(* Logix 5000 project; controller cal1615 1756-L62 rev 20.19; software revision 20.05; part 81 of 81 *)
(* tags used below, declared in another part *)
   A00 : ALIAS FOR hmi_dint[0].0;
   A12 : ALIAS FOR hmi_dint[0].12;
   A30 : ALIAS FOR hmi_dint[0].30;
   accum_filling_on : ALIAS FOR hmi_dint[9].12;
   accum_holding_pressure_on : BOOL;   // Accumulator Holding Pressure Active
   add_sys_ramp : sys_Ramp;   // Addon Ramp
   ai_lpt01_pct : REAL;   // AI: Linear Position Transducer [%]
   ao_prs01 : REAL;   // AO: Pressure 1
   ao_prs02 : REAL;   // AO: Pressure 2
   control_to_empty : ALIAS FOR hmi_dint[9].13;
   di_ss_close_nip : ALIAS FOR p00_io_winder:5:I.14;
   di_ss_nip_auto : ALIAS FOR p00_io_winder:5:I.13;
   do_carriage_lift_sol : ALIAS FOR p00_io_winder:4:O.7;
   do_close_nip_sol : ALIAS FOR p00_io_winder:4:O.8;
   do_nip_illuminated_ss : ALIAS FOR p00_io_winder:4:O.6;
   enable_control : BOOL;   // Accumulator - Enable Control
   filling_pressure : REAL;   // Accumulator Fill Pressure Tare + Tension + Fill PID Offset
   Me : ALIAS FOR p00_wac;
   nip_auto_open_request : BOOL;   // Nip Auto Open Request
   nip_close_request : ALIAS FOR hmi_dint[9].7;
   nip_mode_auto : BOOL;   // Nip Mode Auto
   nip_open_dwell : TIMER;   // Nip Roll Open Dwell Payout must be established before the nip lets go
   nip_open_request : BOOL;   // Nip Open Request
   nip_open_selected : BOOL;   // Nip Selector in OPEN Neither Auto nor Close
   oneshot : DINT;
   param_acc_empty_hyst : REAL;   // Parameter Accumulator Empty Hysteresis Re-engages this far above param_acc_empty_pct so the handover cannot chatter [% o
   param_acc_empty_pct : REAL;   // Parameter Accumulator Empty Pressure bleeds to param_prs_empty and the winder hands back to load cell tension control at
   param_acc_min_limit : REAL;   // Parameter Accumulator Low Min Limimt
   param_accel_rate : REAL;   // Parameter Acceleration Rate
   param_counter_prs : REAL;   // Parameter Counter Pressure
   param_decel_rate : REAL;   // Parameter Decleration Rate
   param_press_slope_empty : REAL;   // Parameter Pressure Curve Slope - BOTH DIRECTIONS Measured on the machine: 62.9 psi gave 30 lbf, 68.0 psi gave 46 lbf (46
   param_prs_empty : REAL;   // Parameter Accumulator Pressure - EMPTY Bled out, carriage on the bottom stop, adds no tension [psi]
   param_prs_fill : REAL;   // Parameter RETIRED - fill pressure is calculated now See filling_pressure [psi]
   param_prs_payout : REAL;   // Parameter RETIRED - payout pressure is calculated now See wac_tension_pressure [psi]
   param_tare_pressure : REAL;   // Parameter Zero-Tension Pressure - PAYING OUT 62.9 - 30/3.14 = 53.4 [psi]
   param_tare_pressure_fill : REAL;   // Parameter Zero-Tension Pressure - FILLING Higher than paying out because friction reverses sign 83 psi held 70 lbf while
   pb_acc_on : ALIAS FOR hmi_dint[9].2;
   request_fill : ALIAS FOR hmi_dint[9].1;
   selected_pressure : REAL;   // Accumulator Selected Tension Pressure
   task_scan_time : REAL;   // Task Scan Time
   task_scan_time_dint : DINT;   // Task Scan
   timer_nip_open_delay : TIMER;   // Nip Open Dwell Timer
   W00 : ALIAS FOR hmi_dint[2].0;
   wac_tension_pressure : REAL;   // Winder Accumulator Tare + Web Tension Pressure Carriage Holds Position at Commanded Tension
   FAULT : BOOL;   // Fault AFI
   HMI : BOOL;   // AFI HMI
   nip_mode_close : BOOL;   // Nip Mode Close
   p00_FlashBit_1Sec : BOOL;   // System Flash Bit 1 Second
   p00_pb_lamp_test : BOOL;
   p00_wac : Accumulator;   // Winder Accumulator
   p00_wac_enabled : BOOL;   // Winder Accumulator Enabled Carriage lift on and pressure commanded Controls which loop holds web tension
   p00_wac_position_pct : REAL;   // Winder Accumulator Carriage Position Filtered [% of Stroke]
   p01_recipe_active : recipe;   // Active Recipe
   p01r09 : routine;   // System Modes
   p01r12_zero_line_speed : BOOL;   // System Line Accel Decel Control Line Speed at Zero
   p29_param_wind_out_stop_pct : REAL;   // Winder Wind Out Stop When the Accumulator Reaches This Position [% of Stroke]
   p29r15_request_run : BOOL;   // Winder Winder A VFD Request Run
   p29r16_request_run : BOOL;   // Winder Winder B VFD Request Run
(* P31_WAC, continued *)

ROUTINE R11_Modes   (* ladder *)
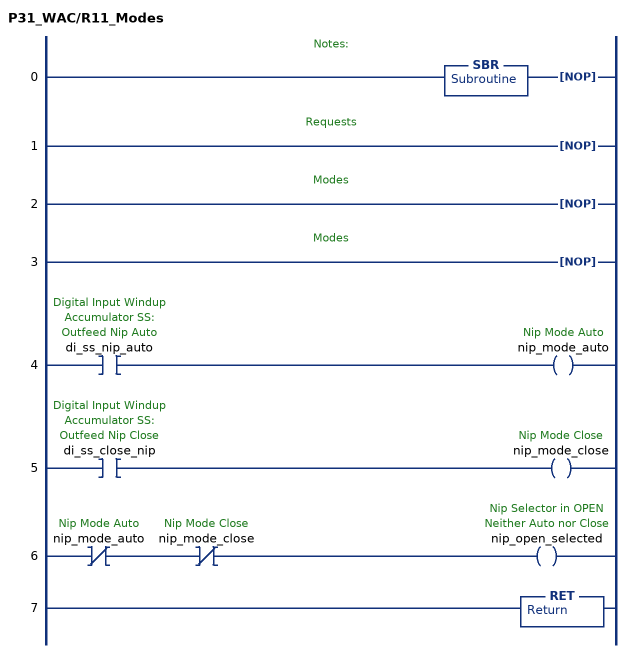
   // Notes:
   0: SBR()NOP();
   // Requests
   1: NOP();
   // Modes
   2: NOP();
   // Modes
   3: NOP();
   4: XIC(di_ss_nip_auto)OTE(nip_mode_auto);
   5: XIC(di_ss_close_nip)OTE(nip_mode_close);
   6: XIO(nip_mode_auto)XIO(nip_mode_close)OTE(nip_open_selected);
   7: RET();
END_ROUTINE

ROUTINE R21_Fill_Request   (* ladder *)
// WAC
// Fill Request and Tension Enable
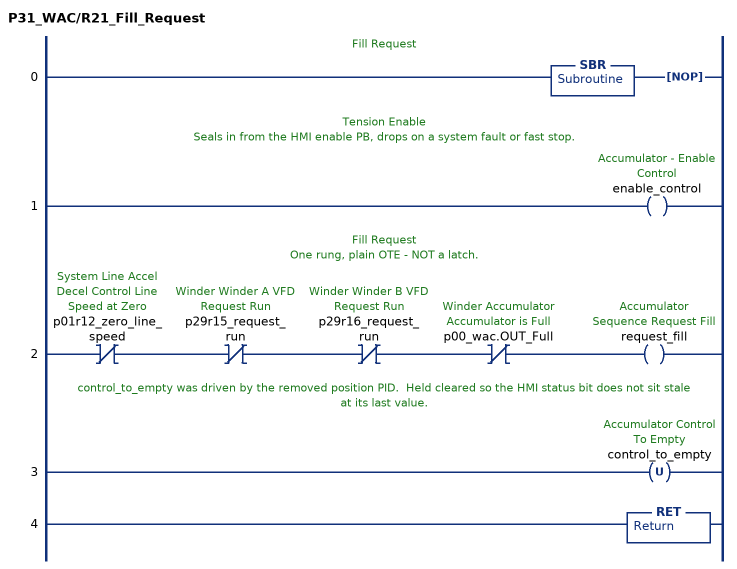
   // Fill Request
   0: SBR()NOP();
   // Tension Enable
   // Seals in from the HMI enable PB, drops on a system fault or fast stop.
   1: OTE(enable_control);
   // Fill Request
   // One rung, plain OTE - NOT a latch.
   2: XIO(p01r12_zero_line_speed)XIO(p29r15_request_run)XIO(p29r16_request_run)XIO(p00_wac.OUT_Full)OTE(request_fill);
   // control_to_empty was driven by the removed position PID.  Held cleared so the HMI status bit does not sit stale at its last value.
   3: OTU(control_to_empty);
   4: RET();
END_ROUTINE

ROUTINE R22_Fill_Pressure   (* ladder *)
// Windup Accumulator
// Fill Pressure
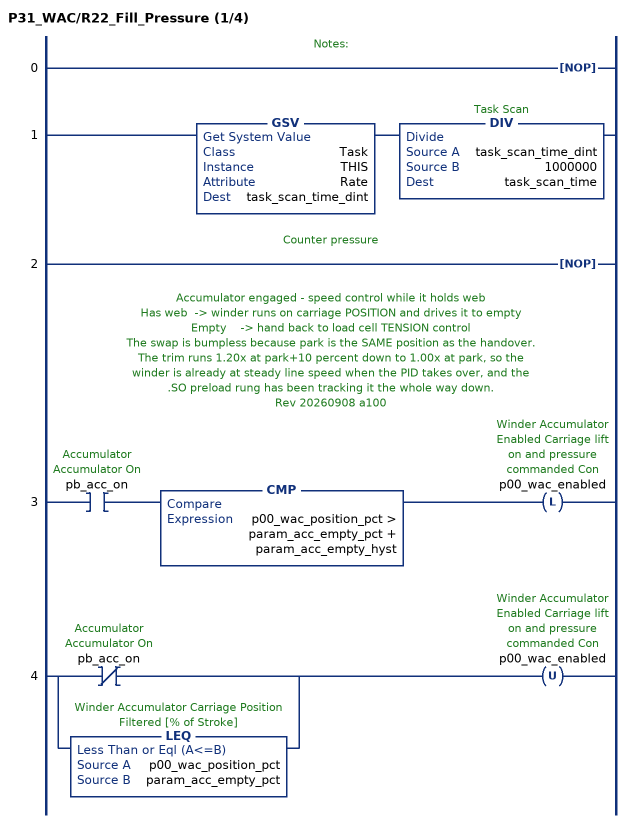
   // Notes:
   0: NOP();
   1: GSV(Task,THIS,Rate,task_scan_time_dint)DIV(task_scan_time_dint,1000000,task_scan_time);
   // Counter pressure
   2: NOP();
   // Accumulator engaged - speed control while it holds web
   // Has web  -> winder runs on carriage POSITION and drives it to empty
   // Empty    -> hand back to load cell TENSION control
   // The swap is bumpless because park is the SAME position as the handover.
   // The trim runs 1.20x at park+10 percent down to 1.00x at park, so the
   // winder is already at steady line speed when the PID takes over, and the
   // .SO preload rung has been tracking it the whole way down.
   // Rev 20260908 a100
   3: XIC(pb_acc_on)CMP(p00_wac_position_pct > param_acc_empty_pct + param_acc_empty_hyst)OTL(p00_wac_enabled);
   4: [XIO(pb_acc_on) ,LEQ(p00_wac_position_pct,param_acc_empty_pct) ]OTU(p00_wac_enabled);
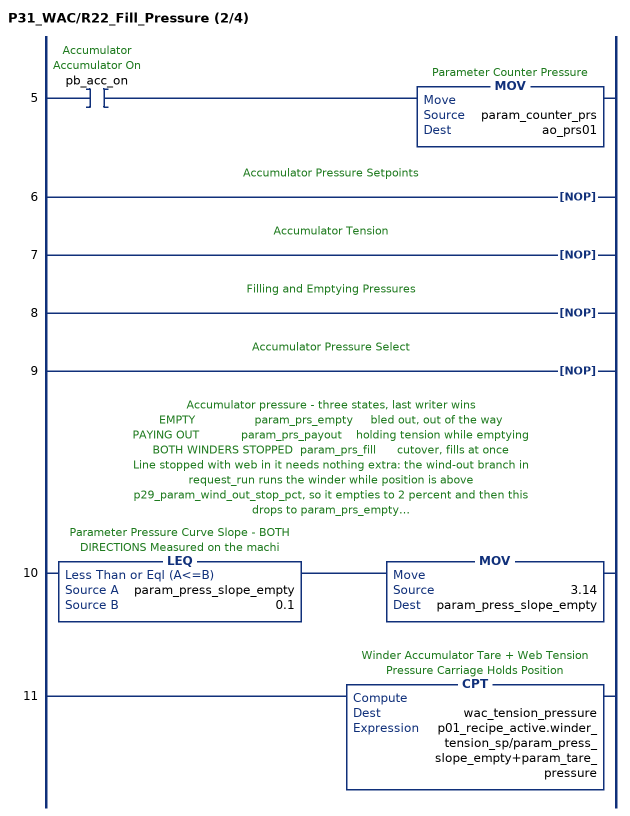
   5: XIC(pb_acc_on)MOV(param_counter_prs,ao_prs01);
   // Accumulator Pressure Setpoints
   6: NOP();
   // Accumulator Tension
   7: NOP();
   // Filling and Emptying Pressures
   8: NOP();
   // Accumulator Pressure Select
   9: NOP();
   // Accumulator pressure - three states, last writer wins
   //   EMPTY                 param_prs_empty     bled out, out of the way
   //   PAYING OUT            param_prs_payout    holding tension while emptying
   //   BOTH WINDERS STOPPED  param_prs_fill      cutover, fills at once
   // Line stopped with web in it needs nothing extra: the wind-out branch in
   // request_run runs the winder while position is above
   // p29_param_wind_out_stop_pct, so it empties to 2 percent and then this
   // drops to param_prs_empty.
   // sys_Ramp below takes every change at param_accel_rate/param_decel_rate,
   // so none of these step.
   // Rev 20260908 a100
   10: LEQ(param_press_slope_empty,0.1)MOV(3.14,param_press_slope_empty);
   11: CPT(wac_tension_pressure,p01_recipe_active.winder_tension_sp/param_press_slope_empty+param_tare_pressure);
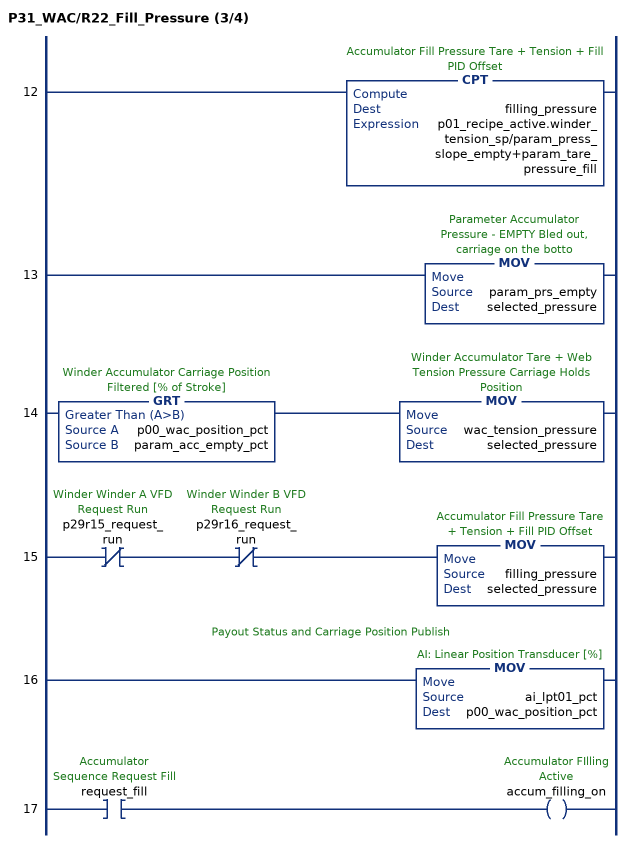
   12: CPT(filling_pressure,p01_recipe_active.winder_tension_sp/param_press_slope_empty+param_tare_pressure_fill);
   13: MOV(param_prs_empty,selected_pressure);
   14: GRT(p00_wac_position_pct,param_acc_empty_pct)MOV(wac_tension_pressure,selected_pressure);
   15: XIO(p29r15_request_run)XIO(p29r16_request_run)MOV(filling_pressure,selected_pressure);
   // Payout Status and Carriage Position Publish
   16: MOV(ai_lpt01_pct,p00_wac_position_pct);
   17: XIC(request_fill)OTE(accum_filling_on);
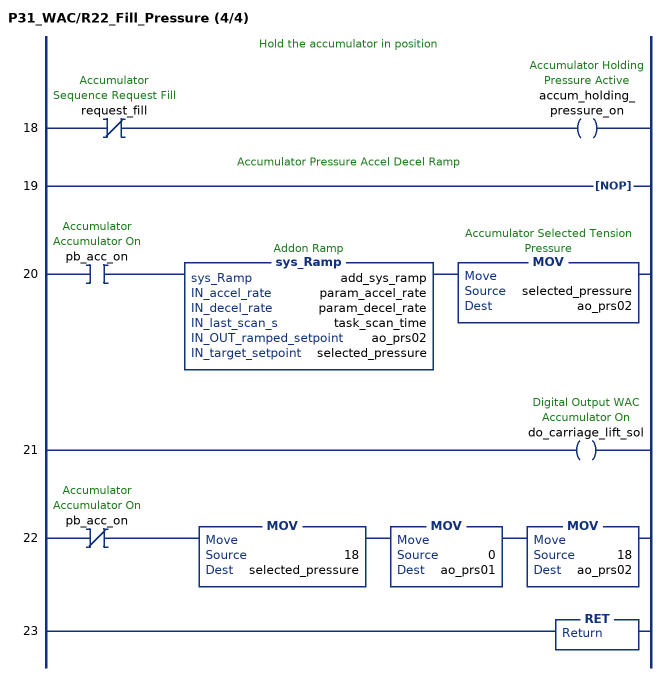
   // Hold the accumulator in position
   18: XIO(request_fill)OTE(accum_holding_pressure_on);
   // Accumulator Pressure Accel Decel Ramp
   19: NOP();
   20: XIC(pb_acc_on)sys_Ramp(add_sys_ramp,param_accel_rate,param_decel_rate,task_scan_time,ao_prs02,selected_pressure)MOV(selected_pressure,ao_prs02);
   21: OTE(do_carriage_lift_sol);
   22: XIO(pb_acc_on)MOV(18,selected_pressure)MOV(0,ao_prs01)MOV(18,ao_prs02);
   23: RET();
END_ROUTINE

ROUTINE R31_Nip_Roll   (* ladder *)
// WAC
// Nip Roll
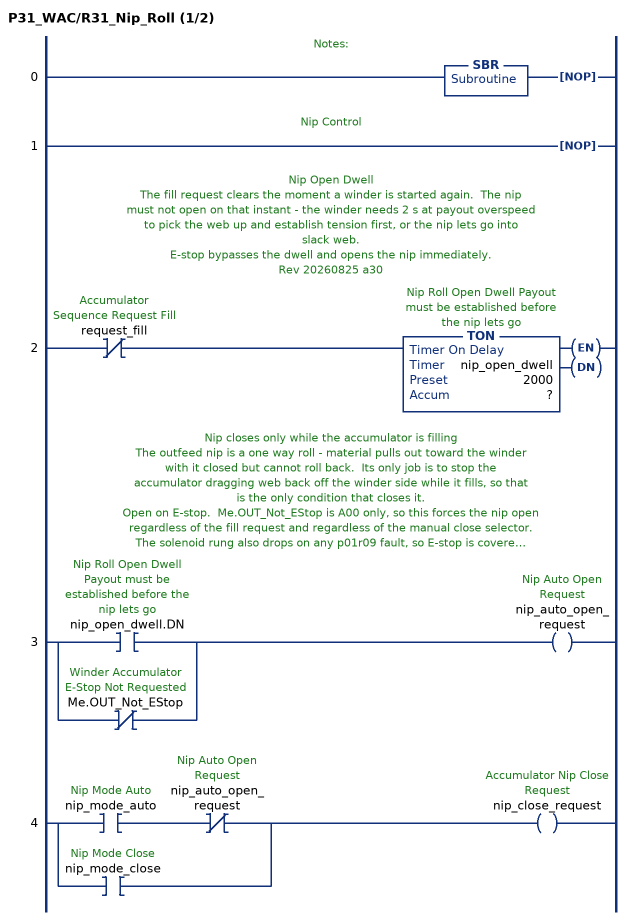
   // Notes:
   0: SBR()NOP();
   // Nip Control
   1: NOP();
   // Nip Open Dwell
   // The fill request clears the moment a winder is started again.  The nip
   // must not open on that instant - the winder needs 2 s at payout overspeed
   // to pick the web up and establish tension first, or the nip lets go into
   // slack web.
   // E-stop bypasses the dwell and opens the nip immediately.
   // Rev 20260825 a30
   2: XIO(request_fill)TON(nip_open_dwell,?,?);
   // Nip closes only while the accumulator is filling
   // The outfeed nip is a one way roll - material pulls out toward the winder
   // with it closed but cannot roll back.  Its only job is to stop the
   // accumulator dragging web back off the winder side while it fills, so that
   // is the only condition that closes it.
   // Open on E-stop.  Me.OUT_Not_EStop is A00 only, so this forces the nip open
   // regardless of the fill request and regardless of the manual close selector.
   // The solenoid rung also drops on any p01r09 fault, so E-stop is covered
   // twice - deliberately.
   // Previously opened on accumulator level above param_acc_min_limit.  That
   // left it open during the fill, which is the one time it needs to be shut.
   // No open delay - the level-based version needed one, this does not.
   // timer_nip_open_delay is left declared and unused.
   // Rev 20260825 a12
   3: [XIC(nip_open_dwell.DN) ,XIO(Me.OUT_Not_EStop) ]OTE(nip_auto_open_request);
   4: [XIC(nip_mode_auto) XIO(nip_auto_open_request) ,XIC(nip_mode_close) ]OTE(nip_close_request);
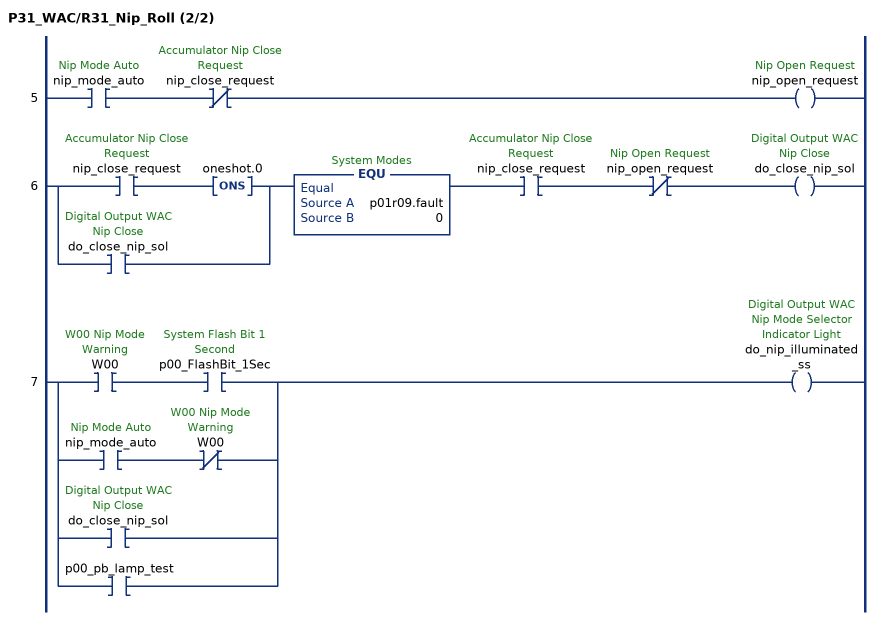
   5: XIC(nip_mode_auto)XIO(nip_close_request)OTE(nip_open_request);
   6: [XIC(nip_close_request) ONS(oneshot.0) ,XIC(do_close_nip_sol) ]EQU(p01r09.fault,0)XIC(nip_close_request)XIO(nip_open_request)OTE(do_close_nip_sol);
   7: [XIC(W00) XIC(p00_FlashBit_1Sec) ,XIC(nip_mode_auto) XIO(W00) ,XIC(do_close_nip_sol) ,XIC(p00_pb_lamp_test) ]OTE(do_nip_illuminated_ss);
END_ROUTINE
END_PROGRAM

PROGRAM ZZZ
END_PROGRAM
